FUNCTION TryConvert_UINT_TO_WORD : BOOL
VAR_INPUT
	in : UINT;
	out : REFERENCE TO WORD;
END_VAR

out := UINT_TO_WORD(in);
TryConvert_UINT_TO_WORD := TRUE;

END_FUNCTION

(* stored: Version 1.1.0.1, ProductVersion 3.1.4024.12
   POU TryConvert_UINT_TO_WORD: Id {64f97b42-8bbb-43a5-960f-5a55d4e73e3a}, SpecialFunc None *)
